RoboDK station: Drillingtask.rdk

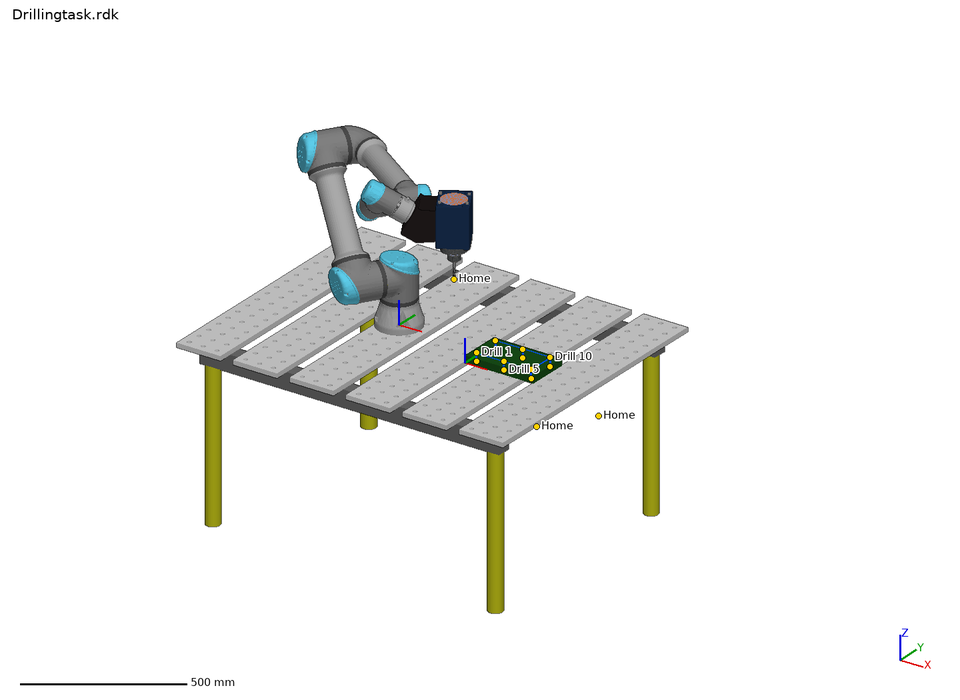
[picture v0: the station drawn from its stored meshes, robots at their saved joint values, targets as dots, program paths as lines]
Station Drillingtask (saved by RoboDK 5.6.3). Poses are relative to the parent item; angles as X-Y-Z fixed-axis rotations.
  - frame UR5e Base at (0, 0, 0) mm
    - robot UR5e: 6 axes, payload 5 kg, reach 850 mm, repeatability 0.03 mm, weight 18.4 kg
        modified DH rows (alpha deg, a mm, theta deg, d mm): 0, 0, 0, 162.5; 90, 0, 180, 0; 0, 425, 0, 0; 0, 392.25, 0, 133.3; -90, 0, 0, 99.7; 90, 0, 180, 99.6
        joint limits [-360, -360, -360, -360, -360, -360] to [360, 360, 360, 360, 360, 360]; home [0, -90, -90, 0, 90, 0]; saved at [-33.011, -48.893, 227.399, -50.338, -219.492, -44.473]
      - tool Custom Spindle, TCP at (0, 119.5, 220.16) mm, rotated rx -60 ry 0 rz 0 deg, size 260.9 x 152 x 222 mm, geometry from Custom Spindle.STEP
    - target Home (joint target) at (275.68, -107.29, 270.75) mm, rotated rx 180 ry 0 rz -60 deg; joints [-33.011, -48.893, 227.399, -50.338, -219.492, -44.473] of UR5e
      - target Home (Cartesian target) at (427.43, -285.95, 271.09) mm, rotated rx 180 ry 0 rz -60 deg; joints [-41.966, -108.916, 291.403, 115.714, -145.435, 123.071] of UR5e
      - target Home (Cartesian target) at (427.43, -285.95, 271.09) mm, rotated rx 180 ry 0 rz -60 deg; joints [-41.966, -108.916, 291.403, 115.714, -145.435, 123.071] of UR5e
      - target Home (Cartesian target) at (427.43, -285.95, 271.09) mm, rotated rx 180 ry 0 rz -60 deg; joints [-41.966, -108.916, 291.403, 115.714, -145.435, 123.071] of UR5e
        - target Home (Cartesian target) at (427.43, -285.95, 271.09) mm, rotated rx 180 ry 0 rz -60 deg; joints [-41.966, -108.916, 291.403, 115.714, -145.435, 123.071] of UR5e
        - target Home (Cartesian target) at (427.43, -285.95, 271.09) mm, rotated rx 180 ry 0 rz -60 deg; joints [-41.966, -108.916, 291.403, 115.714, -145.435, 123.071] of UR5e
  - object Object Table at (120, 0, 0) mm, size 1193.8 x 965.2 x 609.6 mm, geometry from Object Table.wrl
  - frame Frame 2 at (310, -100, 0) mm
    - object Part1 at (0, 0, 0) mm, size 250 x 150 x 25 mm, geometry from Part1.STEP
    - target Drill 1 (Cartesian target) at (25, 25, 30) mm, rotated rx -180 ry 0 rz -60 deg; joints [-16.796, -90.026, 199.263, 30.62, -230.856, -28.029] of UR5e
    - target Drill 2 (Cartesian target) at (25, 25, 1) mm, rotated rx -180 ry 0 rz -60 deg; joints [-16.796, -101.985, 198.011, 43.832, -230.856, -28.029] of UR5e
    - target Drill 3 (Cartesian target) at (25, 25, 30) mm, rotated rx -180 ry 0 rz -60 deg; joints [-16.796, -90.026, 199.263, 30.62, -230.856, -28.029] of UR5e
    - target Drill 4 (Cartesian target) at (125, 25, 30) mm, rotated rx -180 ry 0 rz -60 deg; joints [-10.958, -100.39, 211.32, 31.672, -235.41, -23.461] of UR5e
    - target Drill 5 (Cartesian target) at (125, 25, 1) mm, rotated rx -180 ry 0 rz -60 deg; joints [-10.958, -107.665, 210.6, 39.667, -235.41, -23.461] of UR5e
    - target Drill 6 (Cartesian target) at (125, 25, 30) mm, rotated rx -180 ry 0 rz -60 deg; joints [-10.958, -100.39, 211.32, 31.672, -235.41, -23.461] of UR5e
    - target Drill 7 (Cartesian target) at (225, 25, 30) mm, rotated rx -180 ry 0 rz -60 deg; joints [-8.034, -108.794, 225.016, 27.537, -237.752, -21.361] of UR5e
    - target Drill 8 (Cartesian target) at (225, 25, 1) mm, rotated rx -180 ry 0 rz -60 deg; joints [-8.034, -113.89, 224.507, 33.142, -237.752, -21.361] of UR5e
    - target Drill 9 (Cartesian target) at (225, 25, 30) mm, rotated rx -180 ry 0 rz -60 deg; joints [-8.034, -108.794, 225.016, 27.537, -237.752, -21.361] of UR5e
    - target Drill 10 (Cartesian target) at (225, 125, 30) mm, rotated rx -180 ry 0 rz -60 deg; joints [8.388, -106.918, 220.153, 34.924, -251.399, -11.204] of UR5e
    - target Drill 11 (Cartesian target) at (225, 125, 1) mm, rotated rx -180 ry 0 rz -60 deg; joints [8.388, -112.642, 219.661, 41.141, -251.399, -11.204] of UR5e
    - target Drill 12 (Cartesian target) at (225, 125, 30) mm, rotated rx -180 ry 0 rz -60 deg; joints [8.388, -106.918, 220.153, 34.924, -251.399, -11.204] of UR5e
    - target Drill 13 (Cartesian target) at (125, 125, 30) mm, rotated rx -180 ry 0 rz -60 deg; joints [12.051, -97.893, 204.78, 41.861, -254.521, -9.2] of UR5e
    - target Drill 14 (Cartesian target) at (125, 125, 1) mm, rotated rx -180 ry 0 rz -60 deg; joints [12.051, -107.163, 204.029, 51.882, -254.521, -9.2] of UR5e
    - target Drill 15 (Cartesian target) at (125, 125, 30) mm, rotated rx -180 ry 0 rz -60 deg; joints [12.051, -97.893, 204.78, 41.861, -254.521, -9.2] of UR5e
    - target Drill 16 (Cartesian target) at (25, 125, 30) mm, rotated rx -180 ry 0 rz -60 deg; joints [22.417, -82.428, 188.679, 43.531, -263.438, -3.808] of UR5e
    - target Drill 17 (Cartesian target) at (25, 125, 1) mm, rotated rx -180 ry 0 rz -60 deg; joints [22.417, -112.61, 186.381, 76.011, -263.438, -3.808] of UR5e
    - target Drill 18 (Cartesian target) at (25, 125, 30) mm, rotated rx -180 ry 0 rz -60 deg; joints [22.417, -82.428, 188.679, 43.531, -263.438, -3.808] of UR5e
  - Python program SpindleOff (listed below)
  - Python program SpindleOn (listed below)
  - program Home (4 instructions, listed below)
  - program Prog4 (20 instructions, listed below)
  - program Home (3 instructions, listed below)
  - program MainProgram (3 instructions, listed below)
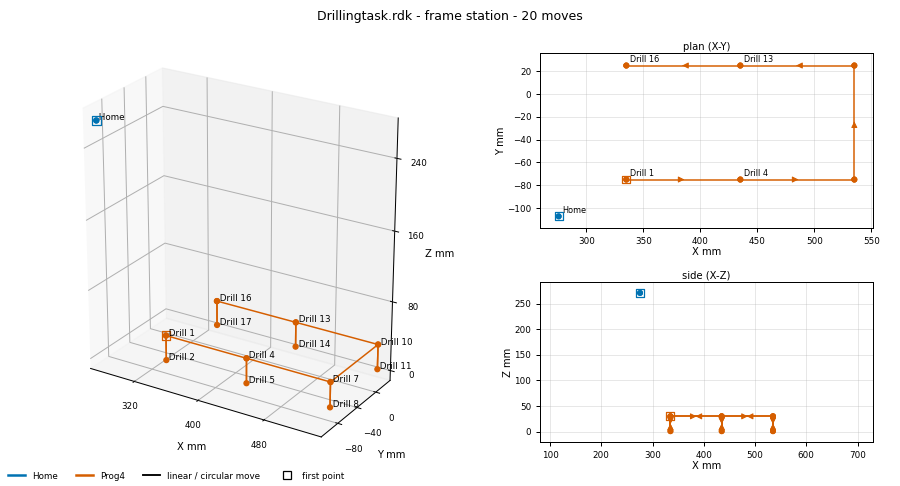
[picture p0: tool path of Drillingtask.rdk in frame station, 20 of 20 moves have a stored position in this frame; points joined in program order, loops and branches not executed]

--- Python program SpindleOff ---
# This script allows adding a trace or a spray deposition
# More information here:
# https://robodk.com/doc/en/PythonAPI/robodk.html#robodk.robolink.Robolink.Spray_Add
#
# Example scripts that use Spray_Add:
#     SpindleOn / SpindleOff    -> Turn trace On/Off
#     ArcOn / ArcOff            -> Turn trace On/Off
#     SprayOn / SprayOff        -> Simulate a spray given a workspace volume (for painting)
#     WeldOn / WeldOff          -> Support for multiple weld guns
#
# Note: Select Esc key or close the RDK project to clear any trace added using this method
# Note: You can pass an ID as first agurment to specify the trace color
#
# Example:
#    SpindleOn(2)           show the trace in blue
#    SpindleOn(red)         show the trace in red
#    SpindleOff             turn off the trace
#
# Note: You can pass the radius of the trace as a second argument
#    SpindleOn(2,2.5)       show the trace in blue with a sphere of radius 2.5 mm
# ---------------------------------------------------------------
#
import sys  # allows getting the passed argument parameters
from robodk.robolink import *  # API to communicate with RoboDK

RDK = Robolink()

# Quit if we are not simulating
if RDK.RunMode() != RUNMODE_SIMULATE:
    quit()

# Stop the trace
RDK.Spray_SetState(SPRAY_OFF)

--- Python program SpindleOn ---
# This script allows adding a trace or a spray deposition
#
# Note: Select Esc key or close the RDK project to clear any trace added using this method
# Note: You can pass an ID as first agurment to specify the trace color
#
# Example:
#    SpindleOn(2)           show the trace in blue
#    SpindleOn(red)         show the trace in red
#    SpindleOff             turn off the trace
#
# Note: You can pass the radius of the trace as a second argument
#    SpindleOn(2,2.5)       show the trace in blue with a sphere of radius 2.5 mm
#
# --------------------------------------------------------------
# This script shows how to create "spray" object in RoboDK that allows simulating particle deposition by using:
# RDK.Spray_Add(tool, object, options_command, volume, geometry)
#    tool: tool item (TCP) to use
#    object: object to project the particles
#    options_command (optional): string to specify options.
#    volume (optional): Matrix of parameters defining the volume of the spray gun
#    geometry (optional): Matrix of vertices defining the triangles.
#
# More information here:
# https://robodk.com/doc/en/PythonAPI/robodk.html#robodk.robolink.Robolink.Spray_Add
# https://robodk.com/doc/en/RoboDK-API.html
#
# The scripts ArcStart, ArcEnd and WeldOn and SpindleOn behave in a similar way, the only difference is the default behavior
# This behavior simmulates Fanuc Arc Welding and triggers appropriate output when using the customized post processor.
# Select ESC to clear the trace manually.
#
# Example scripts that use Spray_Add:
#     SpindleOn / SpindleOff    -> Turn trace On/Off
#     ArcOn / ArcOff            -> Turn trace On/Off
#     SprayOn / SprayOff        -> Simulate a spray given a workspace volume (for painting)
#     WeldOn / WeldOff          -> Support for multiple weld guns

#------------------------------------------------------------------
# Set the tool name as shown in the RoboDK tree (set to None to automatically detect)
TOOL_NAME = None
# TOOL_NAME = "Spindle"

# Set the part name as shown in the RoboDK tree (set to None to automatically detect)
PART_NAME = None
# PART_NAME = "Object"

# Radius of the sphere
SPHERE_RADIUS = 5

# Set the particle color as a named color or as AARRGGBB (alpha channel goes first!)
COLOR = "white"
#COLOR = "green"
#COLOR = "#ffff55bb" # pink-red

# Color list to use if we provide an argument
# Example:
#    SpindleOn(2) will show blue
#    SpindleOn(red) will show red
COLOR_LIST = [COLOR, "red", "green", "blue", "cyan", "magenta", "#ffff55bb"]

#------------------------------------------------------------------
import sys  # allows getting the passed argument parameters
from robodk.robolink import *  # API to communicate with RoboDK

# If an arguments from the object events are provided, retrieve the argument
# (index 0 is the file name)
# Use argument index 1 as color index or named color
if len(sys.argv) >= 2:
    # Use argument 1 as color ID if it is numeric
    arg_1 = sys.argv[1]
    if arg_1.isnumeric():
        color_id = int(arg_1)
        if color_id >= 0:
            color_id = color_id % len(COLOR_LIST)
            COLOR = COLOR_LIST[color_id]
    else:
        # Use the named color (or # color)
        COLOR = arg_1

# Use argument index 2 to set the radius
if len(sys.argv) >= 3:
    # Use argument 1 as color ID if it is numeric
    arg_2 = sys.argv[2]
    try:
        SPHERE_RADIUS = float(arg_2)
    except:
        print("Unable to read paramter 2 as radius")

#------------------------------------------------------------------

# Start the RoboDK API
RDK = Robolink()

# Stop if we are not simulating
if RDK.RunMode() != RUNMODE_SIMULATE:
    quit()

# Create a new spray gun
tool = 0  # auto detect active tool
object = 0  # auto detect object to attach particles

# Use specific tool and part if we provided it
if TOOL_NAME is not None:
    tool = RDK.Item(TOOL_NAME, ITEM_TYPE_TOOL)

if PART_NAME is not None:
    object = RDK.Item(PART_NAME, ITEM_TYPE_OBJECT)

# Create a new object with a spray gun
RDK.Spray_Add(tool, object, "PARTICLE=SPHERE(%.2f) NO_PROJECT COLOR=%s" % (SPHERE_RADIUS, COLOR))  # Do not project
# RDK.Spray_Add(tool, object, "PARTICLE=SPHERE(4) PROJECT") # Project to part
RDK.Spray_SetState(SPRAY_ON)

# Option to use a spread
# coordinates must be provided with respect to the TCP
#close_p0 = [   0,   0, -200] # xyz in mm: Center of the conical ellypse (side 1)
#close_pA = [   5,   0, -200] # xyz in mm: First vertex of the conical ellypse (side 1)
#close_pB = [   0,  10, -200] # xyz in mm: Second vertex of the conical ellypse (side 1)
#close_color = [ 1, 1, 1, 1]  # RGBA (0-1)

#far_p0   = [   0,   0,  50] # xyz in mm: Center of the conical ellypse (side 2)
#far_pA   = [  60,   0,  50] # xyz in mm: First vertex of the conical ellypse (side 2)
#far_pB   = [   0, 120,  50] # xyz in mm: Second vertex of the conical ellypse (side 2)
#far_color   = [ 1, 1, 1, 1]  # RGBA (0-1)

#RDK.Spray_Add(tool, obj, "PARTICLE=CUBE(10,10,2) STEP=8x8")
#RDK.Spray_Add(tool, obj, "PARTICLE=SPHERE(4,8) STEP=8x8")
#RDK.Spray_Add(tool, obj, "PARTICLE=SPHERE(4,8,1,1,0.1) STEP=8x8 RANDX=3")
#RDK.Spray_Add(tool, obj, "PARTICLE=SPHERE(4,8) NO_PROJECT")
#RDK.Spray_Add(tool, obj, "PARTICLE=SPHERE(4,8) STEP=1x0")
#RDK.Spray_Add(tool, obj, "STEP=8x8 RANDX=3", volume.tr(), geom.tr())
#RDK.Spray_SetState(SPRAY_ON)

# Available options:
#     STEP=AxB: Defines the grid to be projected 1x1 means only one line of particle projection (for example, for welding)
#     PARTICLE: Defines the shape and size of particle (sphere or particle), unless a specific geometry is provided:
#       a- SPHERE(radius, facets)
#       b- SPHERE(radius, facets, scalex, scaley, scalez)
#       b- CUBE(sizex, sizey, sizez)
#     RAND=factor: Defines a random factor factor 0 means that the particles are not deposited randomly
#     ELLYPSE: defines the volume as an ellypse (default)
#     RECTANGLE: defines the volume as a rectangle
#     PROJECT: project the particles to the surface (default) (for welding, painting or scanning)
#     NO_PROJECT: does not project the particles to the surface (for example, for 3D printing)

--- program Home (robot UR5e) ---
  Set Ref.: UR5e Base
  Set Tool: Custom Spindle
  MoveL (Home)
  Call Program1

--- program Prog4 (robot UR5e) ---
  Set Ref.: Frame 2
  Set Tool: Custom Spindle
  MoveL (Drill 1)
  MoveL (Drill 2)
  MoveL (Drill 3)
  MoveL (Drill 4)
  MoveL (Drill 5)
  MoveL (Drill 6)
  MoveL (Drill 7)
  MoveL (Drill 8)
  MoveL (Drill 9)
  MoveL (Drill 10)
  MoveL (Drill 11)
  MoveL (Drill 12)
  MoveL (Drill 13)
  MoveL (Drill 14)
  MoveL (Drill 15)
  MoveL (Drill 16)
  MoveL (Drill 17)
  MoveL (Drill 18)

--- program Home (robot UR5e) ---
  Set Ref.: UR5e Base
  Set Tool: Custom Spindle
  MoveL (Home)

--- program MainProgram (robot UR5e) ---
  Call Home
  Call Prog4
  Call Home
